// Mitsubishi GX Works2 project: dataEx05   PLC: Q02/Q02H

PROGRAM MAIN
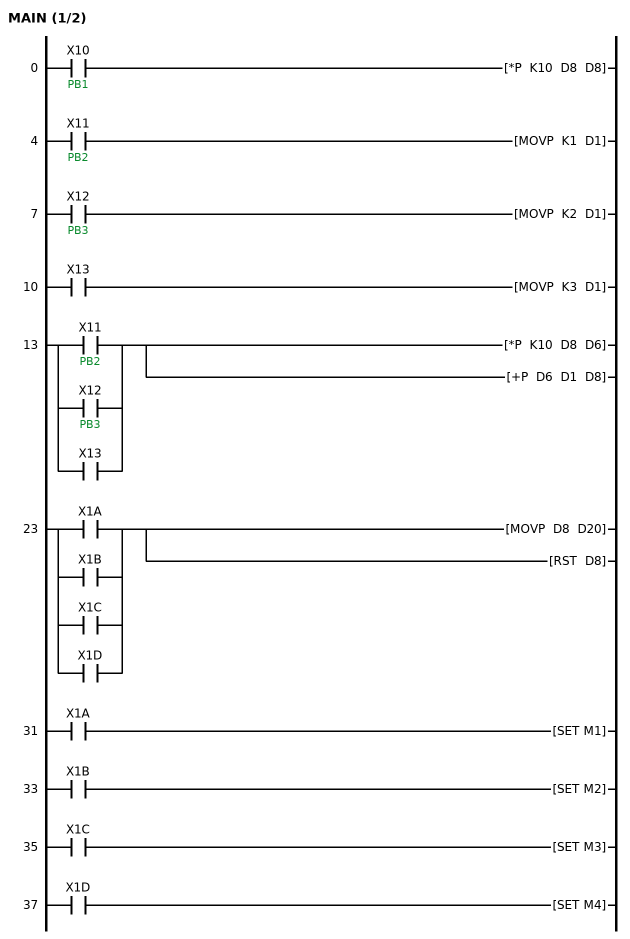
0     LD      X10  ; PB1
      *P      K10 D8 D8
4     LD      X11  ; PB2
      MOVP    K1 D1
7     LD      X12  ; PB3
      MOVP    K2 D1
10    LD      X13
      MOVP    K3 D1
13    LD      X11  ; PB2
      OR      X12  ; PB3
      OR      X13
      *P      K10 D8 D6
      +P      D6 D1 D8
23    LD      X1A
      OR      X1B
      OR      X1C
      OR      X1D
      MOVP    D8 D20
      RST     D8
31    LD      X1A
      SET     M1
33    LD      X1B
      SET     M2
35    LD      X1C
      SET     M3
37    LD      X1D
      SET     M4
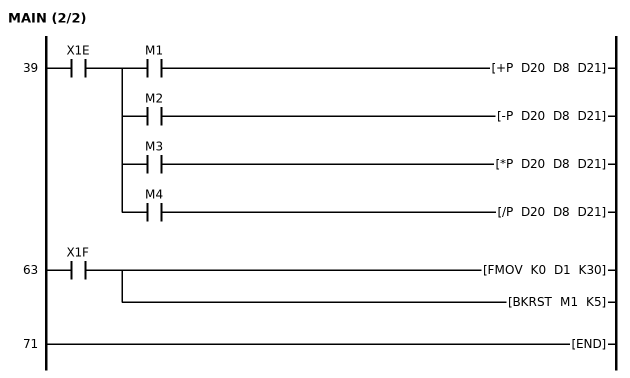
39    LD      X1E
      MPS
      AND     M1
      +P      D20 D8 D21
      MRD
      AND     M2
      -P      D20 D8 D21
      MRD
      AND     M3
      *P      D20 D8 D21
      MPP
      AND     M4
      /P      D20 D8 D21
63    LD      X1F
      FMOV    K0 D1 K30
      BKRST   M1 K5
71    END
END_PROGRAM

// device comments not shown above
X0  ; 공급_후
X1  ; 공급_전
X2  ; 드릴_상
X3  ; 드릴_하
X4  ; 송출_후
X5  ; 송출_전
X6  ; 배출_후
X7  ; 배출_전
X8  ; 매거진
X9  ; 비금속
X0A  ; 금속
Y20  ; 공급_전
Y21  ; 공급_후
Y22  ; 드릴_하강
Y23  ; 송출_전
Y24  ; 송출_후
Y25  ; 배출_전
Y26  ; 배출_후
Y27  ; 컨베어
Y28  ; 가공드
Y29  ; 적색
Y2A  ; 황색
Y2B  ; 녹색
